// TwinCAT 3 PLC project PLC
// ProgramVersion: 3.1.4026.17
// libraries:
//   Tc2_ControllerToolbox, * (Beckhoff Automation GmbH)
//   Tc2_Standard, * (Beckhoff Automation GmbH)
//   Tc2_System, * (Beckhoff Automation GmbH)
// project tree:
//   / PlcTask.TcTTO
//   POUs/ MAIN.TcPOU
// real-time tasks:
//   TASK PlcTask: cycle T#10ms, priority 20, ADS port 350

CONFIGURATION PLC
    RESOURCE PLC ON TwinCAT3
        TASK PlcTask(INTERVAL := T#10ms, PRIORITY := 20);
        PROGRAM MAIN WITH PlcTask : MAIN;
    END_RESOURCE
END_CONFIGURATION

// ---- POUs/MAIN.TcPOU
PROGRAM MAIN
VAR
	//Sinus
	SinusWave	: FB_CTRL_SIGNAL_GENERATOR;
	SinusParams : Tc2_ControllerToolbox.ST_CTRL_SIGNAL_GENERATOR_PARAMS := (tCtrlCycleTime := TIME#10MS, tTaskCycleTime := TIME#10MS, eSignalType := E_CTRL_SIGNAL_TYPE.eCTRL_SINUS, tCylceDuration := TIME#500MS, fAmplitude := 1000);
	SinusSignal : LREAL;

	//Sawtooth
	SawTooth	   : FB_CTRL_SIGNAL_GENERATOR;
	SawToothParams : Tc2_ControllerToolbox.ST_CTRL_SIGNAL_GENERATOR_PARAMS := (tCtrlCycleTime := TIME#10ms, tTaskCycleTime := TIME#10ms, eSignalType := E_CTRL_SIGNAL_TYPE.eCTRL_SAWTOOTH, tCylceDuration := TIME#500ms, fAmplitude := 1000);
	SawToothSignal : LREAL;

	//Triangle
	TriangleWave   : FB_CTRL_SIGNAL_GENERATOR;
	TriangleParams : Tc2_ControllerToolbox.ST_CTRL_SIGNAL_GENERATOR_PARAMS := (tCtrlCycleTime := TIME#10MS, tTaskCycleTime := TIME#10MS, eSignalType := E_CTRL_SIGNAL_TYPE.eCTRL_TRIANGLE, tCylceDuration := TIME#500MS, fAmplitude := 1000);
	TriangleSignal : LREAL;
END_VAR

SinusWave(fManValue :=,
		  eMode		:= E_CTRL_MODE.eCTRL_MODE_ACTIVE,
		  fOut		=> SinusSignal,
		  eState	=>,
		  eErrorId	=>,
		  bError	=>,
		  stParams	:= SinusParams);

SawTooth(fManValue :=,
		 eMode	   := E_CTRL_MODE.eCTRL_MODE_ACTIVE,
		 fOut	   => SawToothSignal,
		 eState	   =>,
		 eErrorId  =>,
		 bError	   =>,
		 stParams  := SawToothParams);

TriangleWave(fManValue :=,
			 eMode	   := E_CTRL_MODE.eCTRL_MODE_ACTIVE,
			 fOut	   => TriangleSignal,
			 eState	   =>,
			 eErrorId  =>,
			 bError	   =>,
			 stParams  := TriangleParams);

END_PROGRAM
